(* Logix 5000 project; controller R5_CSS vendor 1 type 14 code 74 rev 19.11; software revision 19.01; part 12 of 20 *)
(* tags used below, declared in another part *)
   TESTOUT : REAL;
   Bryans_Test_PID : PID;
   PC101A : PRESSURE_CONTROL;   // LOWER QUENCH TOWER PRESSURE TRANSMITTER
   PC101B : PRESSURE_CONTROL;   // UPPER QUENCH TOWER PRESSURE TRANSMITTER PRESSURE CONTOL
   PC134 : PRESSURE_CONTROL;
   PC134_AUTO_Ons : BOOL;
   PC134_AUTO_Ons1 : BOOL;
   PC134_PID : PID;
   PC134_PID_TON : TIMER;
   PC214 : PRESSURE_CONTROL;   // VACUUM SYSTEM PRESSURE TRANSMITTER
   PC214_AUTO_ONS1 : BOOL;
   PC214_MAN_ONS1 : BOOL;
   PC214_PID : PID;   // QUENCH TOWER EXIT PRESSURE CONTROL VALVE
   PC214_PID_PV : REAL;
   PC214_PID_PV_Select : DINT;   // 0 = PT214 1 = PT101A 2 = PT101B
   PC214_PID_TON : TIMER;
   PC271 : PRESSURE_CONTROL;   // VENT HEADER PRESSURE CONTROL
   PC271_AUTO_ONS1 : BOOL;
   PC271_MANUAL_ONS1 : BOOL;
   PC271_PID1 : PID;
   PC271_PID_TON : TIMER;
   PC407A : PRESSURE_CONTROL;   // PRE HX LOW PRESSURE TRANSMITTER
   PC407B : PRESSURE_CONTROL;   // POST HX LOW PRESSURE TRANSMITTER
   Test : INT[500];
   TMR_FAULT : DINT;
(* MainProgram, continued *)

ROUTINE PC134_GTL3_Pressure_PID   (* ladder *)
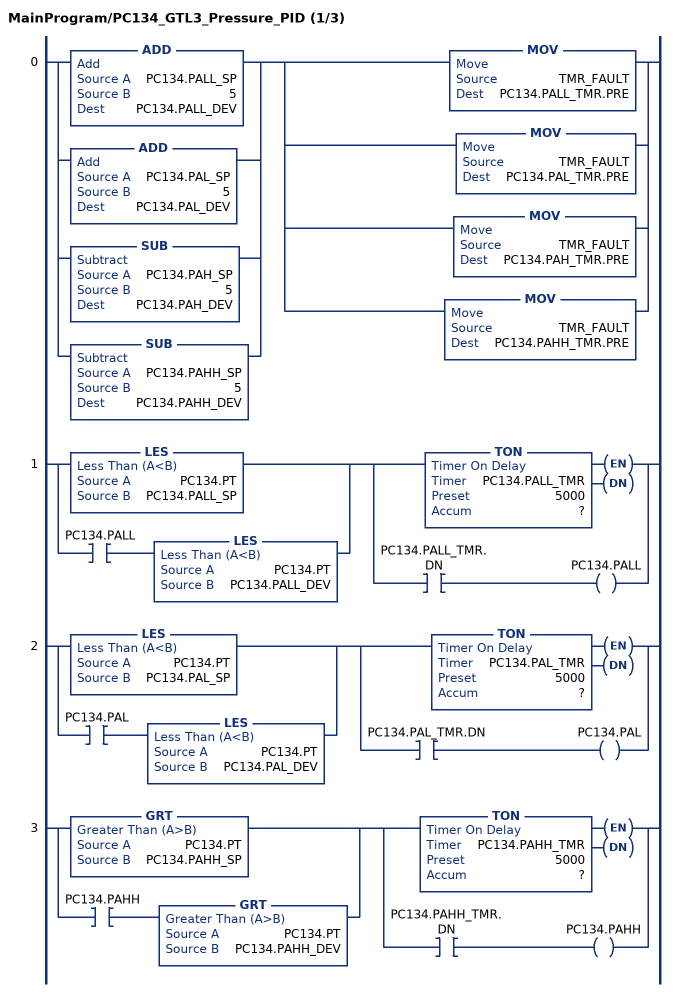
   0: [ADD(PC134.PALL_SP,5,PC134.PALL_DEV) ,ADD(PC134.PAL_SP,5,PC134.PAL_DEV) ,SUB(PC134.PAH_SP,5,PC134.PAH_DEV) ,SUB(PC134.PAHH_SP,5,PC134.PAHH_DEV) ][MOV(TMR_FAULT,PC134.PALL_TMR.PRE) ,MOV(TMR_FAULT,PC134.PAL_TMR.PRE) ,MOV(TMR_FAULT,PC134.PAH_TMR.PRE) ,MOV(TMR_FAULT,PC134.PAHH_TMR.PRE) ];
   1: [LES(PC134.PT,PC134.PALL_SP) ,XIC(PC134.PALL) LES(PC134.PT,PC134.PALL_DEV) ][TON(PC134.PALL_TMR,?,?) ,XIC(PC134.PALL_TMR.DN) OTE(PC134.PALL) ];
   2: [LES(PC134.PT,PC134.PAL_SP) ,XIC(PC134.PAL) LES(PC134.PT,PC134.PAL_DEV) ][TON(PC134.PAL_TMR,?,?) ,XIC(PC134.PAL_TMR.DN) OTE(PC134.PAL) ];
   3: [GRT(PC134.PT,PC134.PAHH_SP) ,XIC(PC134.PAHH) GRT(PC134.PT,PC134.PAHH_DEV) ][TON(PC134.PAHH_TMR,?,?) ,XIC(PC134.PAHH_TMR.DN) OTE(PC134.PAHH) ];
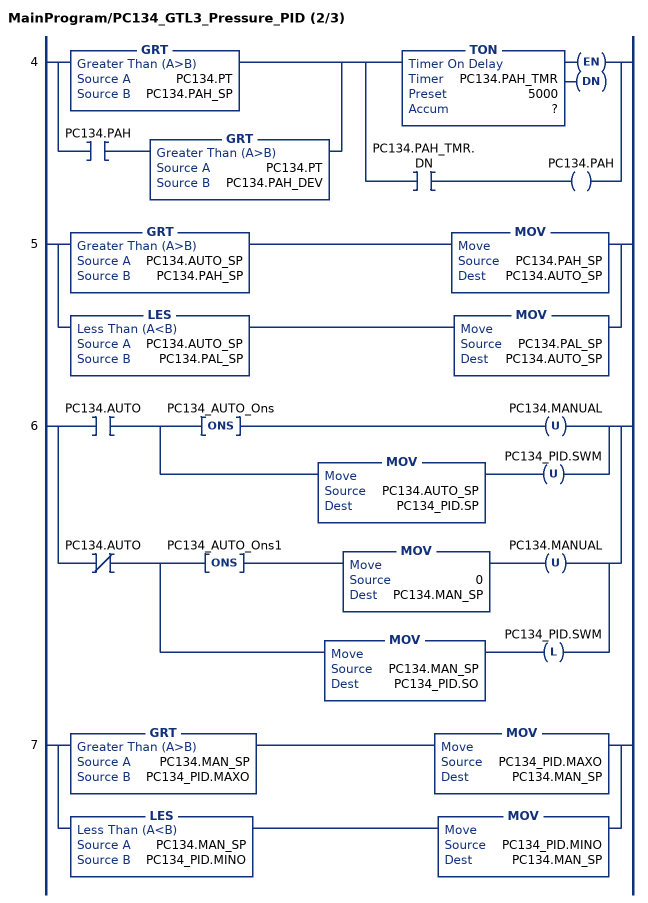
   4: [GRT(PC134.PT,PC134.PAH_SP) ,XIC(PC134.PAH) GRT(PC134.PT,PC134.PAH_DEV) ][TON(PC134.PAH_TMR,?,?) ,XIC(PC134.PAH_TMR.DN) OTE(PC134.PAH) ];
   5: [GRT(PC134.AUTO_SP,PC134.PAH_SP) MOV(PC134.PAH_SP,PC134.AUTO_SP) ,LES(PC134.AUTO_SP,PC134.PAL_SP) MOV(PC134.PAL_SP,PC134.AUTO_SP) ];
   6: [XIC(PC134.AUTO) [ONS(PC134_AUTO_Ons) OTU(PC134.MANUAL) ,MOV(PC134.AUTO_SP,PC134_PID.SP) OTU(PC134_PID.SWM) ] ,XIO(PC134.AUTO) [ONS(PC134_AUTO_Ons1) MOV(0,PC134.MAN_SP) OTU(PC134.MANUAL) ,MOV(PC134.MAN_SP,PC134_PID.SO) OTL(PC134_PID.SWM) ] ];
   7: [GRT(PC134.MAN_SP,PC134_PID.MAXO) MOV(PC134_PID.MAXO,PC134.MAN_SP) ,LES(PC134.MAN_SP,PC134_PID.MINO) MOV(PC134_PID.MINO,PC134.MAN_SP) ];
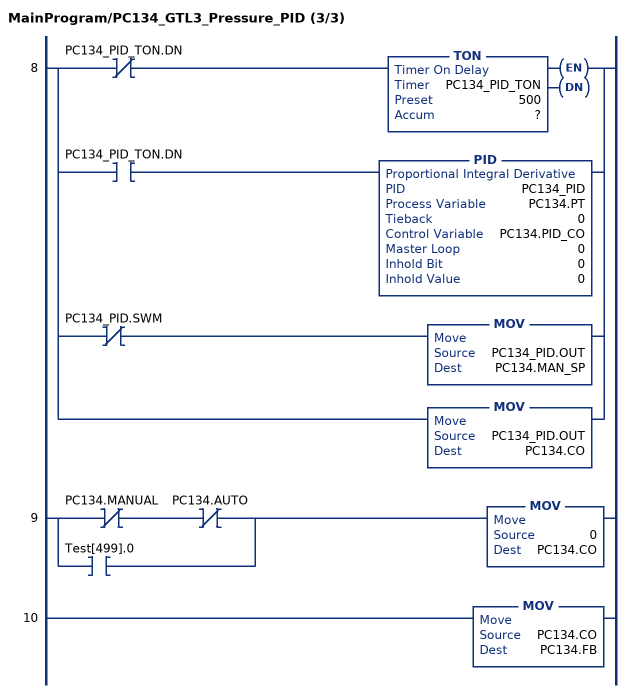
   8: [XIO(PC134_PID_TON.DN) TON(PC134_PID_TON,?,?) ,XIC(PC134_PID_TON.DN) PID(PC134_PID,PC134.PT,0,PC134.PID_CO,0,0,0) ,XIO(PC134_PID.SWM) MOV(PC134_PID.OUT,PC134.MAN_SP) ,MOV(PC134_PID.OUT,PC134.CO) ];
   9: [XIO(PC134.MANUAL) XIO(PC134.AUTO) ,XIC(Test[499].0) ]MOV(0,PC134.CO);
   10: MOV(PC134.CO,PC134.FB);
END_ROUTINE

ROUTINE PC214_VacuumControl   (* ladder *)
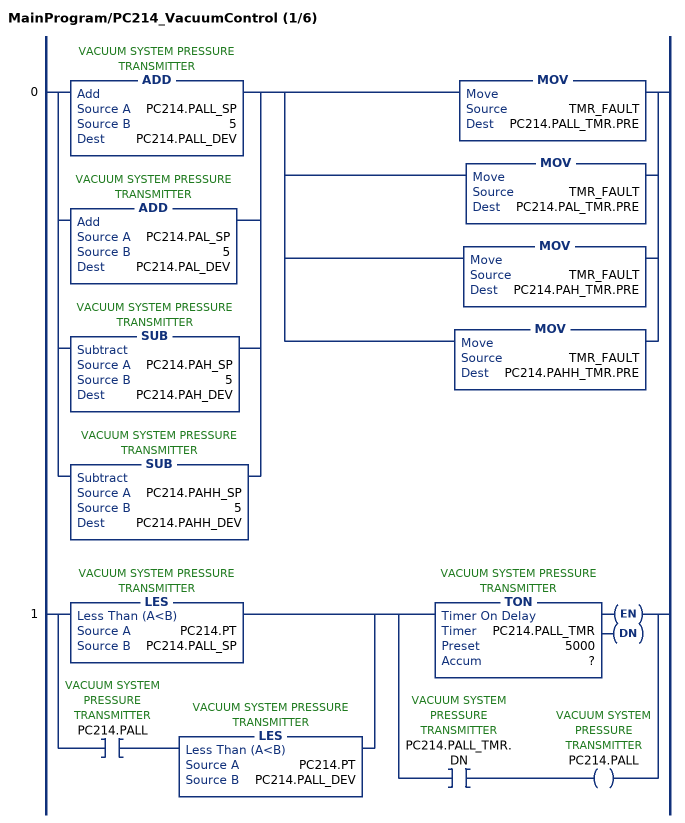
   0: [ADD(PC214.PALL_SP,5,PC214.PALL_DEV) ,ADD(PC214.PAL_SP,5,PC214.PAL_DEV) ,SUB(PC214.PAH_SP,5,PC214.PAH_DEV) ,SUB(PC214.PAHH_SP,5,PC214.PAHH_DEV) ][MOV(TMR_FAULT,PC214.PALL_TMR.PRE) ,MOV(TMR_FAULT,PC214.PAL_TMR.PRE) ,MOV(TMR_FAULT,PC214.PAH_TMR.PRE) ,MOV(TMR_FAULT,PC214.PAHH_TMR.PRE) ];
   1: [LES(PC214.PT,PC214.PALL_SP) ,XIC(PC214.PALL) LES(PC214.PT,PC214.PALL_DEV) ][TON(PC214.PALL_TMR,?,?) ,XIC(PC214.PALL_TMR.DN) OTE(PC214.PALL) ];
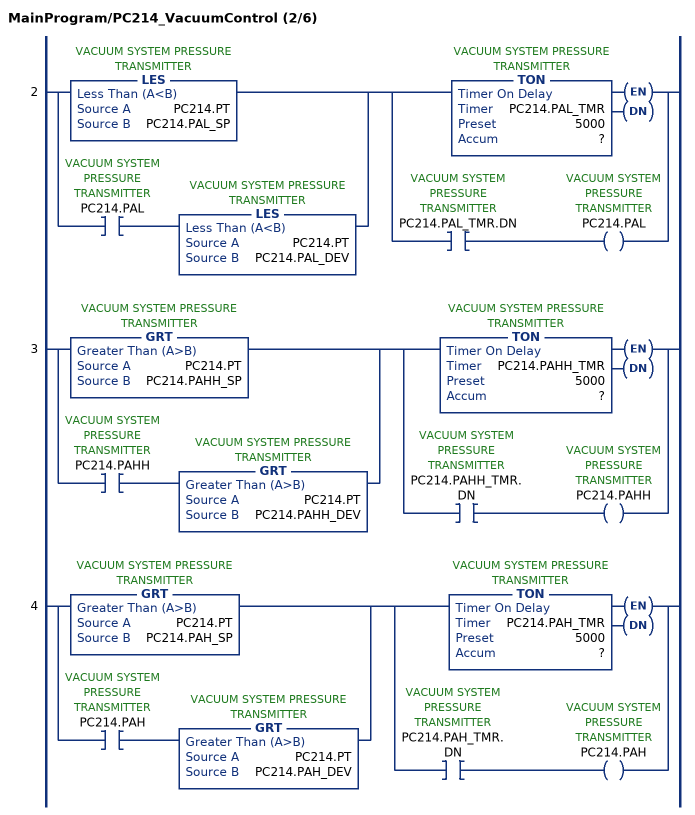
   2: [LES(PC214.PT,PC214.PAL_SP) ,XIC(PC214.PAL) LES(PC214.PT,PC214.PAL_DEV) ][TON(PC214.PAL_TMR,?,?) ,XIC(PC214.PAL_TMR.DN) OTE(PC214.PAL) ];
   3: [GRT(PC214.PT,PC214.PAHH_SP) ,XIC(PC214.PAHH) GRT(PC214.PT,PC214.PAHH_DEV) ][TON(PC214.PAHH_TMR,?,?) ,XIC(PC214.PAHH_TMR.DN) OTE(PC214.PAHH) ];
   4: [GRT(PC214.PT,PC214.PAH_SP) ,XIC(PC214.PAH) GRT(PC214.PT,PC214.PAH_DEV) ][TON(PC214.PAH_TMR,?,?) ,XIC(PC214.PAH_TMR.DN) OTE(PC214.PAH) ];
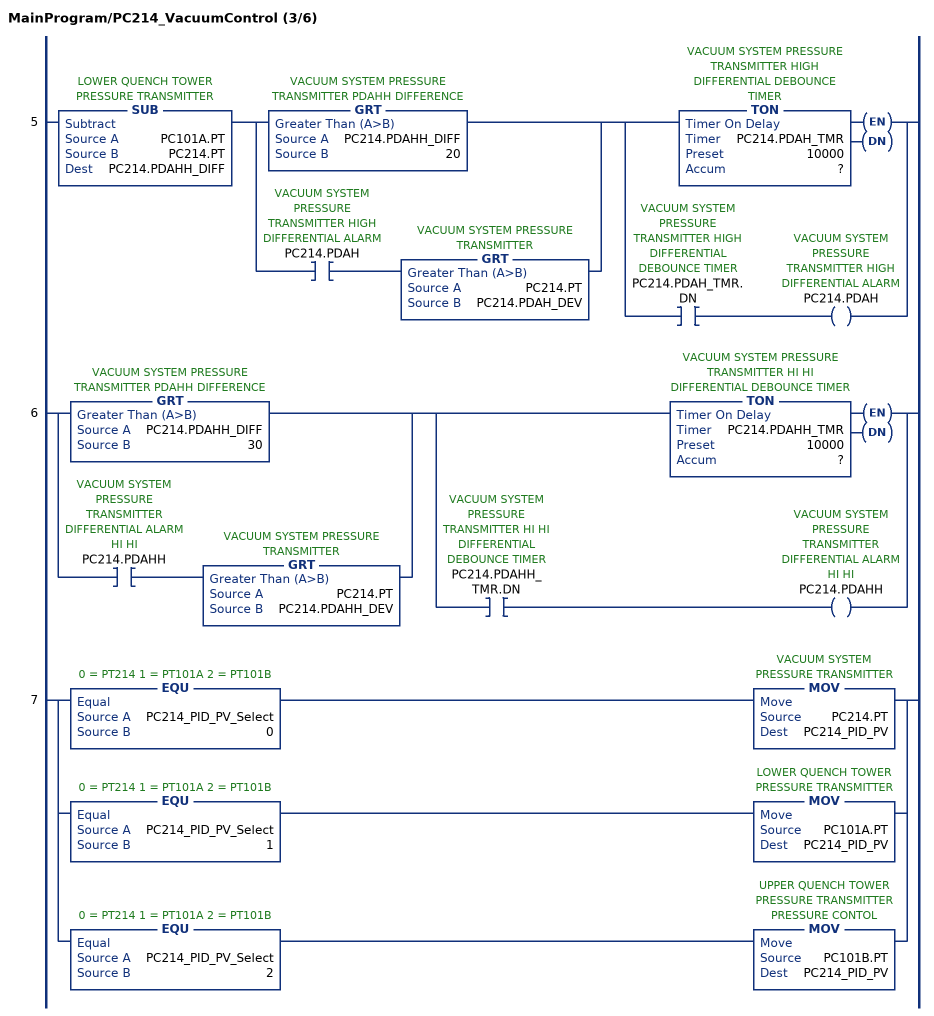
   5: SUB(PC101A.PT,PC214.PT,PC214.PDAHH_DIFF)[GRT(PC214.PDAHH_DIFF,20) ,XIC(PC214.PDAH) GRT(PC214.PT,PC214.PDAH_DEV) ][TON(PC214.PDAH_TMR,?,?) ,XIC(PC214.PDAH_TMR.DN) OTE(PC214.PDAH) ];
   6: [GRT(PC214.PDAHH_DIFF,30) ,XIC(PC214.PDAHH) GRT(PC214.PT,PC214.PDAHH_DEV) ][TON(PC214.PDAHH_TMR,?,?) ,XIC(PC214.PDAHH_TMR.DN) OTE(PC214.PDAHH) ];
   7: [EQU(PC214_PID_PV_Select,0) MOV(PC214.PT,PC214_PID_PV) ,EQU(PC214_PID_PV_Select,1) MOV(PC101A.PT,PC214_PID_PV) ,EQU(PC214_PID_PV_Select,2) MOV(PC101B.PT,PC214_PID_PV) ];
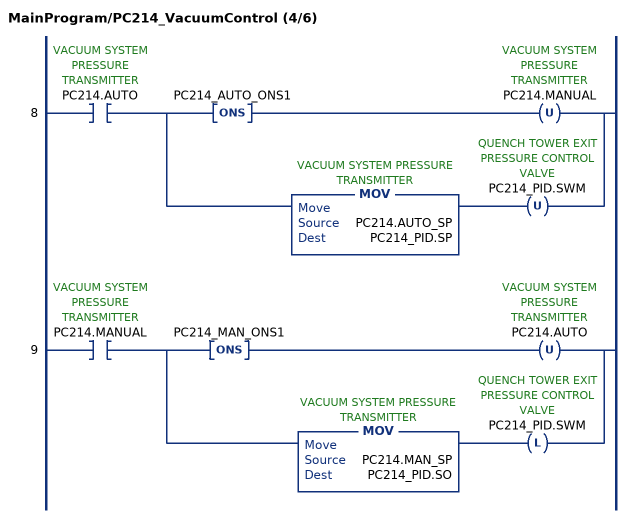
   8: XIC(PC214.AUTO)[ONS(PC214_AUTO_ONS1) OTU(PC214.MANUAL) ,MOV(PC214.AUTO_SP,PC214_PID.SP) OTU(PC214_PID.SWM) ];
   9: XIC(PC214.MANUAL)[ONS(PC214_MAN_ONS1) OTU(PC214.AUTO) ,MOV(PC214.MAN_SP,PC214_PID.SO) OTL(PC214_PID.SWM) ];
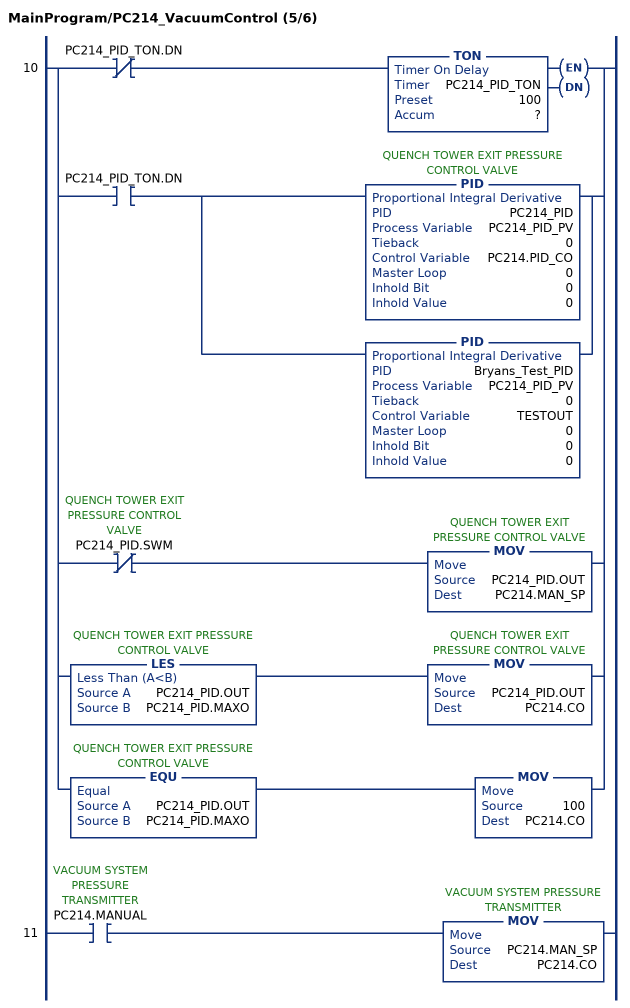
   10: [XIO(PC214_PID_TON.DN) TON(PC214_PID_TON,?,?) ,XIC(PC214_PID_TON.DN) [PID(PC214_PID,PC214_PID_PV,0,PC214.PID_CO,0,0,0) ,PID(Bryans_Test_PID,PC214_PID_PV,0,TESTOUT,0,0,0) ] ,XIO(PC214_PID.SWM) MOV(PC214_PID.OUT,PC214.MAN_SP) ,LES(PC214_PID.OUT,PC214_PID.MAXO) MOV(PC214_PID.OUT,PC214.CO) ,EQU(PC214_PID.OUT,PC214_PID.MAXO) MOV(100,PC214.CO) ];
   11: XIC(PC214.MANUAL)MOV(PC214.MAN_SP,PC214.CO);
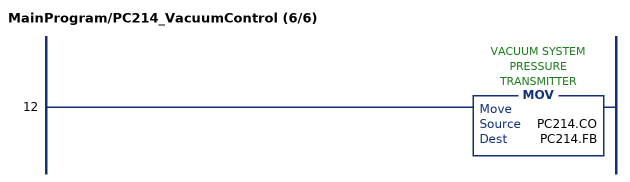
   12: MOV(PC214.CO,PC214.FB);
END_ROUTINE

ROUTINE PC271_CoalesceTankVentPress_PID   (* ladder *)
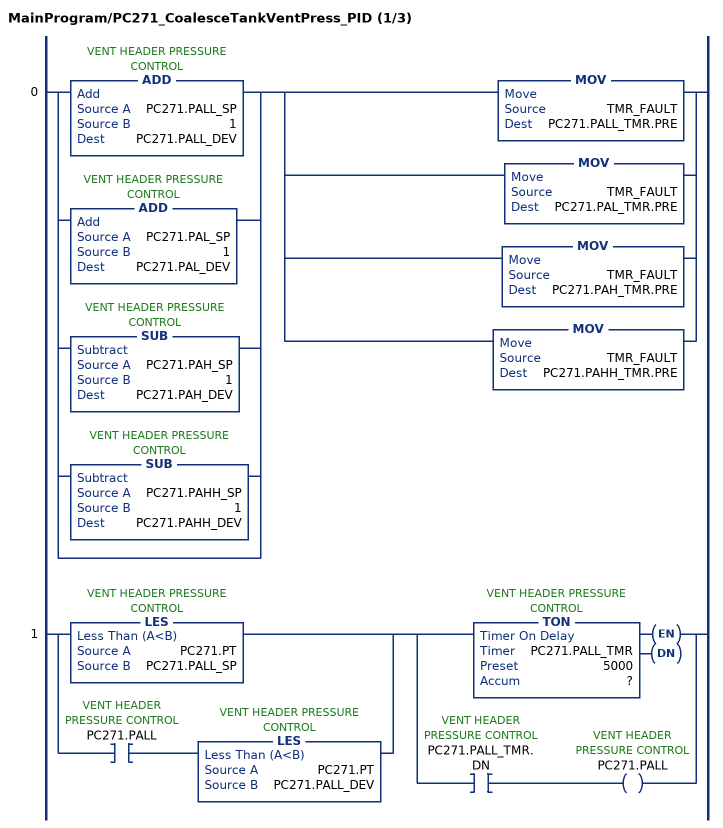
   0: [ADD(PC271.PALL_SP,1,PC271.PALL_DEV) ,ADD(PC271.PAL_SP,1,PC271.PAL_DEV) ,SUB(PC271.PAH_SP,1,PC271.PAH_DEV) ,SUB(PC271.PAHH_SP,1,PC271.PAHH_DEV) ,][MOV(TMR_FAULT,PC271.PALL_TMR.PRE) ,MOV(TMR_FAULT,PC271.PAL_TMR.PRE) ,MOV(TMR_FAULT,PC271.PAH_TMR.PRE) ,MOV(TMR_FAULT,PC271.PAHH_TMR.PRE) ];
   1: [LES(PC271.PT,PC271.PALL_SP) ,XIC(PC271.PALL) LES(PC271.PT,PC271.PALL_DEV) ][TON(PC271.PALL_TMR,?,?) ,XIC(PC271.PALL_TMR.DN) OTE(PC271.PALL) ];
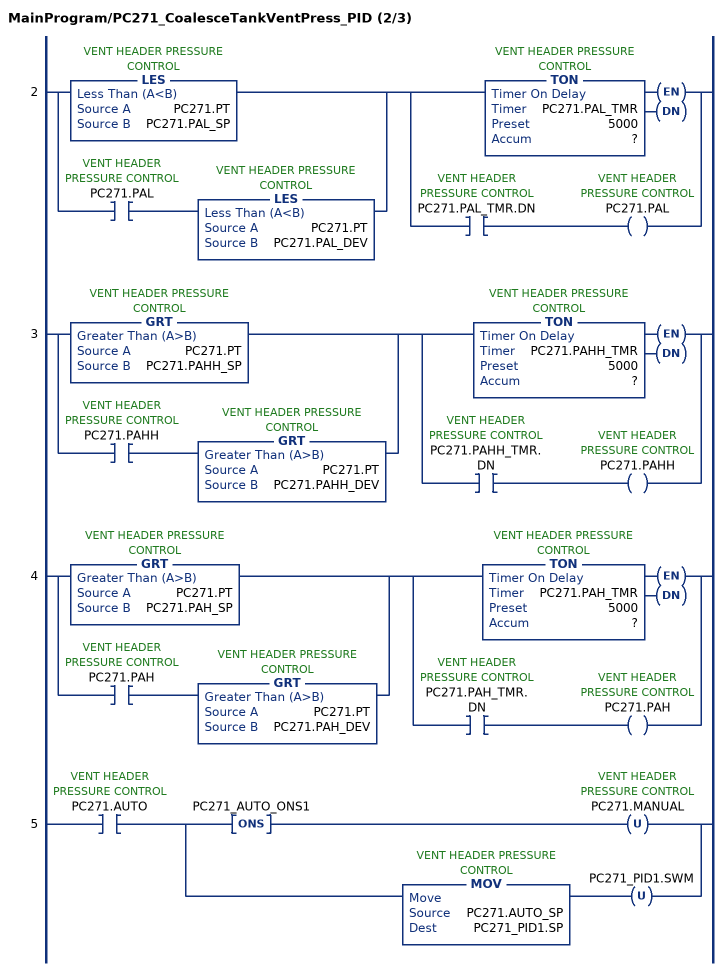
   2: [LES(PC271.PT,PC271.PAL_SP) ,XIC(PC271.PAL) LES(PC271.PT,PC271.PAL_DEV) ][TON(PC271.PAL_TMR,?,?) ,XIC(PC271.PAL_TMR.DN) OTE(PC271.PAL) ];
   3: [GRT(PC271.PT,PC271.PAHH_SP) ,XIC(PC271.PAHH) GRT(PC271.PT,PC271.PAHH_DEV) ][TON(PC271.PAHH_TMR,?,?) ,XIC(PC271.PAHH_TMR.DN) OTE(PC271.PAHH) ];
   4: [GRT(PC271.PT,PC271.PAH_SP) ,XIC(PC271.PAH) GRT(PC271.PT,PC271.PAH_DEV) ][TON(PC271.PAH_TMR,?,?) ,XIC(PC271.PAH_TMR.DN) OTE(PC271.PAH) ];
   5: XIC(PC271.AUTO)[ONS(PC271_AUTO_ONS1) OTU(PC271.MANUAL) ,MOV(PC271.AUTO_SP,PC271_PID1.SP) OTU(PC271_PID1.SWM) ];
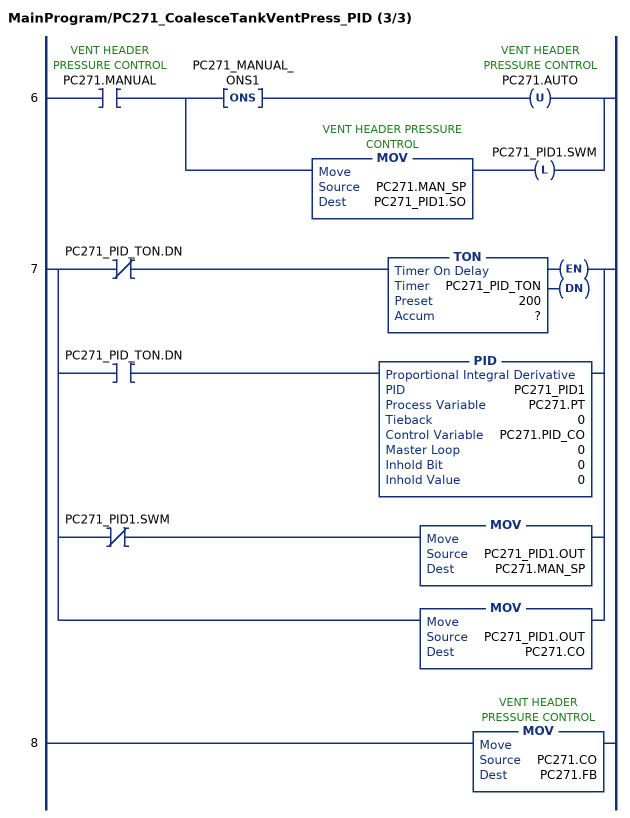
   6: XIC(PC271.MANUAL)[ONS(PC271_MANUAL_ONS1) OTU(PC271.AUTO) ,MOV(PC271.MAN_SP,PC271_PID1.SO) OTL(PC271_PID1.SWM) ];
   7: [XIO(PC271_PID_TON.DN) TON(PC271_PID_TON,?,?) ,XIC(PC271_PID_TON.DN) PID(PC271_PID1,PC271.PT,0,PC271.PID_CO,0,0,0) ,XIO(PC271_PID1.SWM) MOV(PC271_PID1.OUT,PC271.MAN_SP) ,MOV(PC271_PID1.OUT,PC271.CO) ];
   8: MOV(PC271.CO,PC271.FB);
END_ROUTINE

ROUTINE PC407A_PreFilterPressure   (* ladder *)
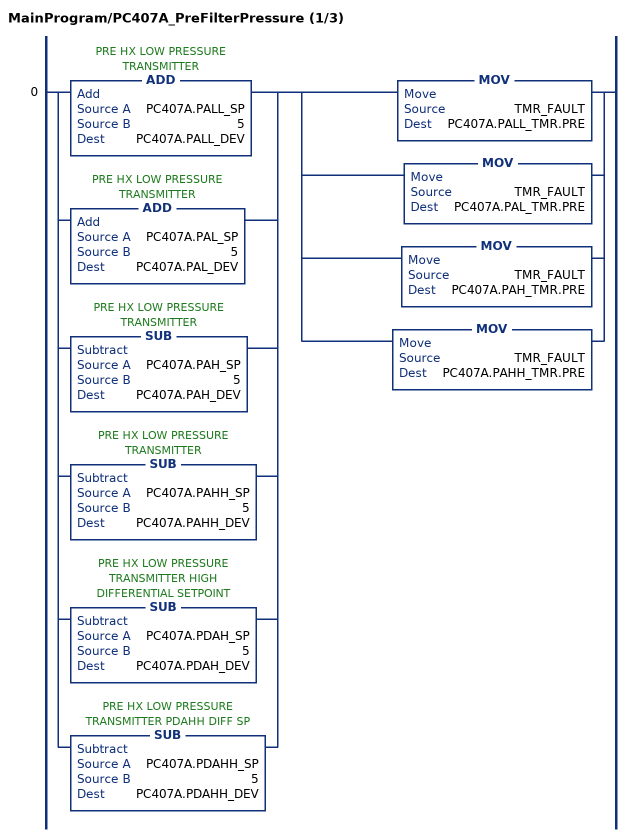
   0: [ADD(PC407A.PALL_SP,5,PC407A.PALL_DEV) ,ADD(PC407A.PAL_SP,5,PC407A.PAL_DEV) ,SUB(PC407A.PAH_SP,5,PC407A.PAH_DEV) ,SUB(PC407A.PAHH_SP,5,PC407A.PAHH_DEV) ,SUB(PC407A.PDAH_SP,5,PC407A.PDAH_DEV) ,SUB(PC407A.PDAHH_SP,5,PC407A.PDAHH_DEV) ][MOV(TMR_FAULT,PC407A.PALL_TMR.PRE) ,MOV(TMR_FAULT,PC407A.PAL_TMR.PRE) ,MOV(TMR_FAULT,PC407A.PAH_TMR.PRE) ,MOV(TMR_FAULT,PC407A.PAHH_TMR.PRE) ];
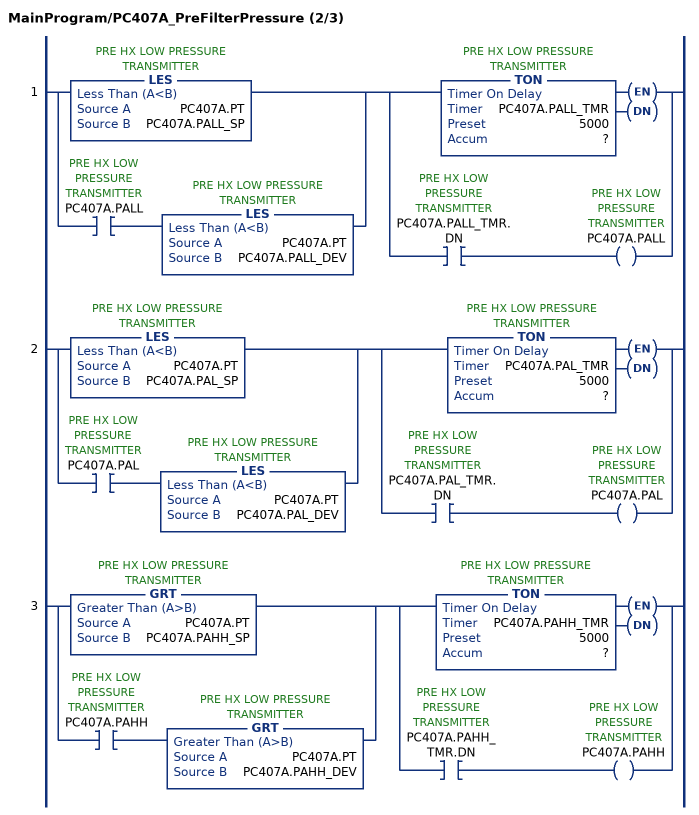
   1: [LES(PC407A.PT,PC407A.PALL_SP) ,XIC(PC407A.PALL) LES(PC407A.PT,PC407A.PALL_DEV) ][TON(PC407A.PALL_TMR,?,?) ,XIC(PC407A.PALL_TMR.DN) OTE(PC407A.PALL) ];
   2: [LES(PC407A.PT,PC407A.PAL_SP) ,XIC(PC407A.PAL) LES(PC407A.PT,PC407A.PAL_DEV) ][TON(PC407A.PAL_TMR,?,?) ,XIC(PC407A.PAL_TMR.DN) OTE(PC407A.PAL) ];
   3: [GRT(PC407A.PT,PC407A.PAHH_SP) ,XIC(PC407A.PAHH) GRT(PC407A.PT,PC407A.PAHH_DEV) ][TON(PC407A.PAHH_TMR,?,?) ,XIC(PC407A.PAHH_TMR.DN) OTE(PC407A.PAHH) ];
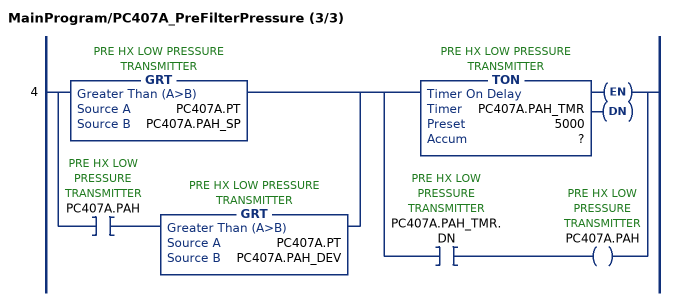
   4: [GRT(PC407A.PT,PC407A.PAH_SP) ,XIC(PC407A.PAH) GRT(PC407A.PT,PC407A.PAH_DEV) ][TON(PC407A.PAH_TMR,?,?) ,XIC(PC407A.PAH_TMR.DN) OTE(PC407A.PAH) ];
END_ROUTINE

ROUTINE PC407B_PostFilterPressure   (* ladder *)
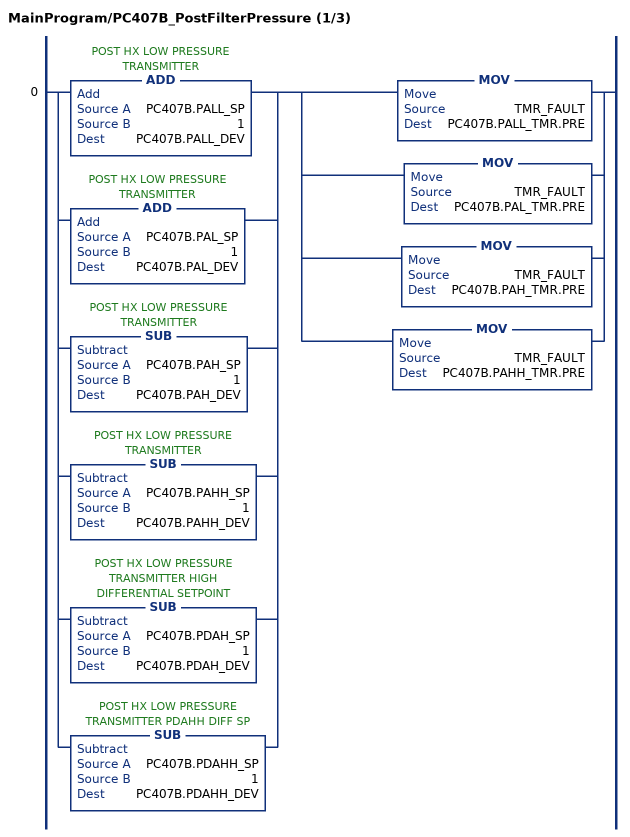
   0: [ADD(PC407B.PALL_SP,1,PC407B.PALL_DEV) ,ADD(PC407B.PAL_SP,1,PC407B.PAL_DEV) ,SUB(PC407B.PAH_SP,1,PC407B.PAH_DEV) ,SUB(PC407B.PAHH_SP,1,PC407B.PAHH_DEV) ,SUB(PC407B.PDAH_SP,1,PC407B.PDAH_DEV) ,SUB(PC407B.PDAHH_SP,1,PC407B.PDAHH_DEV) ][MOV(TMR_FAULT,PC407B.PALL_TMR.PRE) ,MOV(TMR_FAULT,PC407B.PAL_TMR.PRE) ,MOV(TMR_FAULT,PC407B.PAH_TMR.PRE) ,MOV(TMR_FAULT,PC407B.PAHH_TMR.PRE) ];
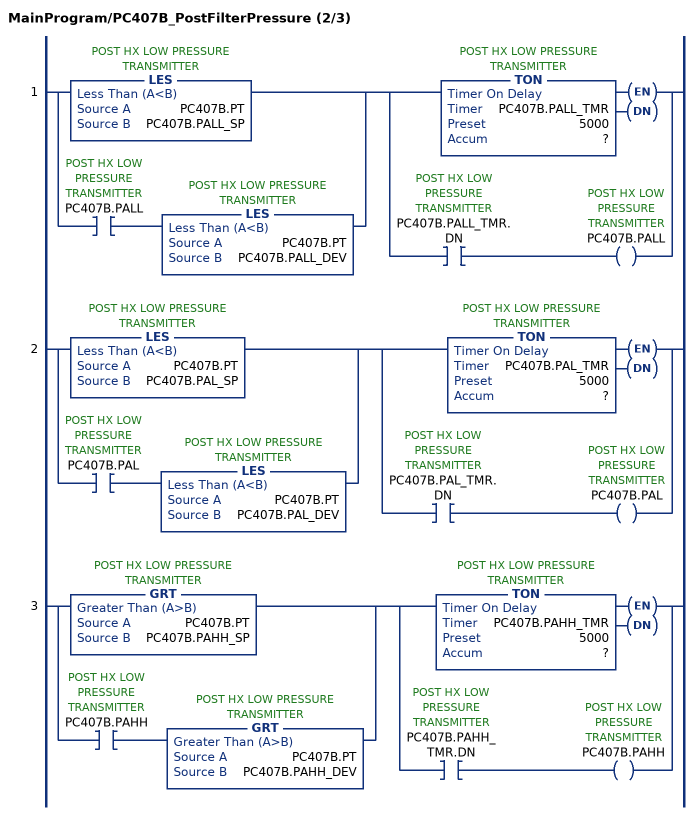
   1: [LES(PC407B.PT,PC407B.PALL_SP) ,XIC(PC407B.PALL) LES(PC407B.PT,PC407B.PALL_DEV) ][TON(PC407B.PALL_TMR,?,?) ,XIC(PC407B.PALL_TMR.DN) OTE(PC407B.PALL) ];
   2: [LES(PC407B.PT,PC407B.PAL_SP) ,XIC(PC407B.PAL) LES(PC407B.PT,PC407B.PAL_DEV) ][TON(PC407B.PAL_TMR,?,?) ,XIC(PC407B.PAL_TMR.DN) OTE(PC407B.PAL) ];
   3: [GRT(PC407B.PT,PC407B.PAHH_SP) ,XIC(PC407B.PAHH) GRT(PC407B.PT,PC407B.PAHH_DEV) ][TON(PC407B.PAHH_TMR,?,?) ,XIC(PC407B.PAHH_TMR.DN) OTE(PC407B.PAHH) ];
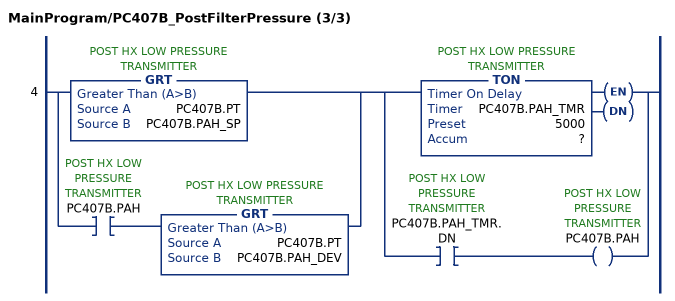
   4: [GRT(PC407B.PT,PC407B.PAH_SP) ,XIC(PC407B.PAH) GRT(PC407B.PT,PC407B.PAH_DEV) ][TON(PC407B.PAH_TMR,?,?) ,XIC(PC407B.PAH_TMR.DN) OTE(PC407B.PAH) ];
END_ROUTINE
